// TIA Portal V20 export
FUNCTION "NodeStatusAlarms" : Void   // FC19, LAD
BEGIN

REGION Network 1
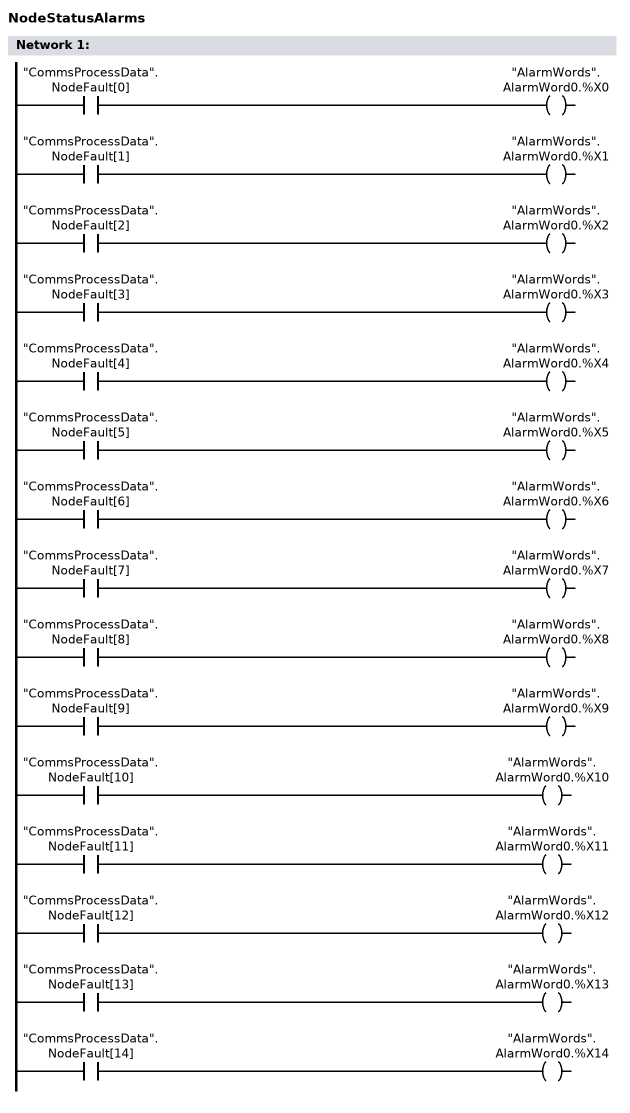
   RUNG wire#powerrail
      Contact( "CommsProcessData".NodeFault[0] )
      Coil( "AlarmWords".AlarmWord0.%X0 )
   END_RUNG
   RUNG wire#powerrail
      Contact( "CommsProcessData".NodeFault[1] )
      Coil( "AlarmWords".AlarmWord0.%X1 )
   END_RUNG
   RUNG wire#powerrail
      Contact( "CommsProcessData".NodeFault[2] )
      Coil( "AlarmWords".AlarmWord0.%X2 )
   END_RUNG
   RUNG wire#powerrail
      Contact( "CommsProcessData".NodeFault[3] )
      Coil( "AlarmWords".AlarmWord0.%X3 )
   END_RUNG
   RUNG wire#powerrail
      Contact( "CommsProcessData".NodeFault[4] )
      Coil( "AlarmWords".AlarmWord0.%X4 )
   END_RUNG
   RUNG wire#powerrail
      Contact( "CommsProcessData".NodeFault[5] )
      Coil( "AlarmWords".AlarmWord0.%X5 )
   END_RUNG
   RUNG wire#powerrail
      Contact( "CommsProcessData".NodeFault[6] )
      Coil( "AlarmWords".AlarmWord0.%X6 )
   END_RUNG
   RUNG wire#powerrail
      Contact( "CommsProcessData".NodeFault[7] )
      Coil( "AlarmWords".AlarmWord0.%X7 )
   END_RUNG
   RUNG wire#powerrail
      Contact( "CommsProcessData".NodeFault[8] )
      Coil( "AlarmWords".AlarmWord0.%X8 )
   END_RUNG
   RUNG wire#powerrail
      Contact( "CommsProcessData".NodeFault[9] )
      Coil( "AlarmWords".AlarmWord0.%X9 )
   END_RUNG
   RUNG wire#powerrail
      Contact( "CommsProcessData".NodeFault[10] )
      Coil( "AlarmWords".AlarmWord0.%X10 )
   END_RUNG
   RUNG wire#powerrail
      Contact( "CommsProcessData".NodeFault[11] )
      Coil( "AlarmWords".AlarmWord0.%X11 )
   END_RUNG
   RUNG wire#powerrail
      Contact( "CommsProcessData".NodeFault[12] )
      Coil( "AlarmWords".AlarmWord0.%X12 )
   END_RUNG
   RUNG wire#powerrail
      Contact( "CommsProcessData".NodeFault[13] )
      Coil( "AlarmWords".AlarmWord0.%X13 )
   END_RUNG
   RUNG wire#powerrail
      Contact( "CommsProcessData".NodeFault[14] )
      Coil( "AlarmWords".AlarmWord0.%X14 )
   END_RUNG
   // the same network as SCL:
   "AlarmWords".AlarmWord0.%X0 := "CommsProcessData".NodeFault[0];
   "AlarmWords".AlarmWord0.%X1 := "CommsProcessData".NodeFault[1];
   "AlarmWords".AlarmWord0.%X2 := "CommsProcessData".NodeFault[2];
   "AlarmWords".AlarmWord0.%X3 := "CommsProcessData".NodeFault[3];
   "AlarmWords".AlarmWord0.%X4 := "CommsProcessData".NodeFault[4];
   "AlarmWords".AlarmWord0.%X5 := "CommsProcessData".NodeFault[5];
   "AlarmWords".AlarmWord0.%X6 := "CommsProcessData".NodeFault[6];
   "AlarmWords".AlarmWord0.%X7 := "CommsProcessData".NodeFault[7];
   "AlarmWords".AlarmWord0.%X8 := "CommsProcessData".NodeFault[8];
   "AlarmWords".AlarmWord0.%X9 := "CommsProcessData".NodeFault[9];
   "AlarmWords".AlarmWord0.%X10 := "CommsProcessData".NodeFault[10];
   "AlarmWords".AlarmWord0.%X11 := "CommsProcessData".NodeFault[11];
   "AlarmWords".AlarmWord0.%X12 := "CommsProcessData".NodeFault[12];
   "AlarmWords".AlarmWord0.%X13 := "CommsProcessData".NodeFault[13];
   "AlarmWords".AlarmWord0.%X14 := "CommsProcessData".NodeFault[14];
END_REGION
END_FUNCTION
